// TIA Portal V20 export
ORGANIZATION_BLOCK "Main"   // OB1, LAD, ProgramCycle
TITLE = "Main Program Sweep (Cycle)"
{ S7_Optimized_Access := 'TRUE' }
// stored: SetENOAutomatically false
   VAR_INPUT
      Initial_Call : Bool;   // Initial call of this OB
      Remanence : Bool;   // =True, if remanent data are available
   END_VAR
   VAR_TEMP   // added for the SCL form of the ladder/FBD networks
      _w1 : Bool;
   END_VAR
BEGIN

REGION Network 1
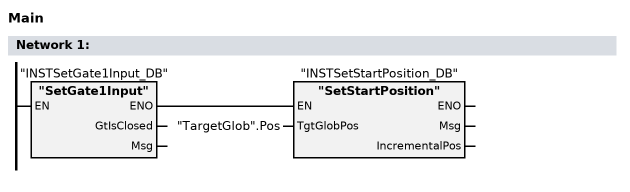
   RUNG wire#powerrail
      "INSTSetGate1Input_DB"(GtIsClosed =>, Msg =>)
      "INSTSetStartPosition_DB"(TgtGlobPos := "TargetGlob".Pos, Msg =>, IncrementalPos =>)
   END_RUNG
   // the same network as SCL:
   "INSTSetGate1Input_DB"(ENO => #_w1);   // "SetGate1Input"
   IF #_w1 THEN
       "INSTSetStartPosition_DB"(TgtGlobPos := "TargetGlob".Pos);   // "SetStartPosition"
   END_IF;
END_REGION
END_ORGANIZATION_BLOCK
